FUNCTION_BLOCK Undefined_State IMPLEMENTS ITF_State
VAR_INPUT
END_VAR
VAR_OUTPUT
END_VAR
VAR
	pPML_Base : POINTER TO PML_StatePattern_Base;
	_stateMachine : IPmlStateMachine;
END_VAR

METHOD Cycle : BOOL
VAR_INPUT
END_VAR
IF _stateMachine.GetCurrentState() = E_PMLState.ePMLState_Aborting THEN
	pPML_Base^.SetState(pPML_Base^.aborting);
END_IF
END_METHOD

METHOD FB_init : BOOL
VAR_INPUT
	bInitRetains : BOOL; // if TRUE, the retain variables are initialized (warm start / cold start)
	bInCopyCode : BOOL;  // if TRUE, the instance afterwards gets moved into the copy code (online change)
	pPML_Base : POINTER TO PML_StatePattern_Base;
	statemachine : IPmlStateMachine;
END_VAR
_stateMachine := statemachine;
THIS^.pPML_Base := pPML_Base;
END_METHOD

END_FUNCTION_BLOCK

(* stored: Version 1.1.0.1, ProductVersion 3.1.4024.11
   POU Undefined_State: Id {c5bff6b1-4064-4b65-bcf0-b9e64e1cfe6a}, SpecialFunc None
   Method Cycle: Id {aa642894-c26f-4e32-a785-c0387e3cb65b}
   Method FB_init: Id {eaa13123-eaab-4247-803b-a53ca19725f9} *)
